TYPE st_AllocateCircleMoveStructure :
STRUCT
	Latch : LREAL;
	Position :LREAL;
//	Excute	:BOOL;
//	Done	 :BOOL;
//	Busy  : BOOL;
//	Occupied : BOOL;	
	HandShake					: st_HandshakeBase;
END_STRUCT
END_TYPE

(* stored: Version 1.1.0.1, ProductVersion 3.1.4024.13
   DUT st_AllocateCircleMoveStructure: Id {7d850219-e82e-467e-a484-5565d783e4a8} *)
